Staubli VAL3: setAllBlend.pgx

public program setAllBlend(num x_nNewValue, num x_nOldValue)
  local num i
  local num l_nSize
  local TrajectoryItem l_tTraj
begin
  // check if is OK
  if x_nNewValue!=x_nOldValue
    // get the size
    call trajType:getSizeItem(false,l_nSize)
    for i=0 to (l_nSize-1)
      // get it
      call trajType:getTrajItem(l_tTraj,i)
      // check it
      if l_tTraj.nom_speed.leave==x_nOldValue or (l_tTraj.nom_speed.blend==off and x_nOldValue==-1)
        if x_nNewValue<0
          l_tTraj.nom_speed.blend=off
        else
          l_tTraj.nom_speed.leave=l_tTraj.nom_speed.reach=x_nNewValue
          l_tTraj.nom_speed.blend=joint
        endIf
      endIf
      // set it
      call trajType:setTrajItem(l_tTraj,i)
    endFor
  endIf
end
